{attribute 'linkalways'} 
{attribute 'no_explicit_call' := 'This FB is a CLASS and must be accessed using methods or properties'}
{attribute 'enable_dynamic_creation'}
FUNCTION_BLOCK OutputPort EXTENDS Disposable IMPLEMENTS I_OutputPort
VAR
	_name : T_MAXSTRING;
	_data : I_Datatype;
	parent : I_HaveOutputPorts;
	eventEmitter : EventEmitter;
END_VAR

METHOD PUBLIC Accept
VAR_INPUT
	Visitor : I_OutputPortVisitor;
END_VAR
Visitor.VisitOutputPort(this^);
END_METHOD

PROPERTY PUBLIC Data : I_Datatype
GET
Data := _data;
END_GET
END_PROPERTY

METHOD Protected EmitOnOutputPortChangeEvent
VAR_INPUT
	PortChanged : I_OutputPort;
END_VAR
VAR
	pOutputPortChangeEvent : POINTER TO OutputPortChangedEvent;
END_VAR
pOutputPortChangeEvent := __NEW(OutputPortChangedEvent(TargetOutputPort := PortChanged));
eventEmitter.Emit('OnOutputPortChanged',pOutputPortChangeEvent^);
pOutputPortChangeEvent^.Dispose();
END_METHOD

METHOD FB_init : BOOL
VAR_INPUT
	bInitRetains : BOOL; // if TRUE, the retain variables are initialized (warm start / cold start)
	bInCopyCode : BOOL;  // if TRUE, the instance afterwards gets moved into the copy code (online change)
	Name : T_MAXSTRING;
	Data : I_Datatype;
	Parent : I_HaveOutputPorts;
END_VAR
_name := Name;
_data := Data;
RegisterWithParent(Parent);
END_METHOD

PROPERTY PUBLIC Name : T_MAXSTRING
GET
Name := _name;
END_GET
END_PROPERTY

METHOD PUBLIC OffEvent
VAR_INPUT
	EventName : T_MaxString;
	EventHandler : I_EventHandler;
END_VAR
eventEmitter.OffEvent(EventName, EventHandler);
END_METHOD

METHOD PUBLIC OnceEvent
VAR_INPUT
	EventName : T_MaxString;
	EventHandler : I_EventHandler;
END_VAR
eventEmitter.OnceEvent(EventName, EventHandler);
END_METHOD

METHOD PUBLIC OnEvent
VAR_INPUT
	EventName : T_MaxString;
	EventHandler : I_EventHandler;
END_VAR
eventEmitter.OnEvent(EventName, EventHandler);
END_METHOD

METHOD PUBLIC RegisterWithParent
VAR_INPUT
	Parent : I_HaveOutputPorts;
END_VAR
IF Parent = 0 THEN
	RETURN;
END_IF

THIS^.parent := Parent;
Parent.AddOutputPort(THIS^);
END_METHOD

METHOD PUBLIC SerializeWith
VAR_INPUT
	Serializer : I_Serializer;
END_VAR
Serializer.StartObject();
Serializer.AddKeyString('name',_name);
Serializer.Addkey('datatype');
_data.SerializeTypeWith(Serializer);
Serializer.AddkeyObject('value',_data);
Serializer.EndObject();
END_METHOD

END_FUNCTION_BLOCK

(* stored: Version 1.1.0.1, ProductVersion 3.1.4024.12
   POU OutputPort: Id {4c7e0bce-9eb0-0f6a-044f-6a3cfc8b783d}, SpecialFunc None
   Folder Constructor: Id {677256cd-e8af-081b-2804-5689f5f4149b}
   Folder Protected: Id {6f5f4b13-ef19-01e5-075e-0ea3b801d3d7}
   Method Accept: Id {685a8b40-a5b2-0491-3a06-acbf37dad5a1}
   Property Data: Id {f88ed905-c54b-4c6d-be97-9339266743b0}
   Get Get: Id {120b55e4-6686-441d-ae9a-fc15e5629d7f}
   Method EmitOnOutputPortChangeEvent: Id {4cedd9f2-3d84-035e-18ce-b7ebc3af2524}
   Method FB_init: Id {1ba1d2d7-341d-0e8e-05ef-f5346255db4e}
   Property Name: Id {a6251d93-37b5-06d7-00eb-bc1261f23075}
   Get Get: Id {66530c4b-9811-0535-0d83-3db73e2195f3}
   Method OffEvent: Id {5f0c98a6-efae-06ce-0d53-00d24017a360}
   Method OnceEvent: Id {33aa55e6-cc64-0804-1f68-fe127e9ffd59}
   Method OnEvent: Id {83584882-e2df-000f-0211-5ef5ee02b990}
   Method RegisterWithParent: Id {c7baf534-bf05-4f66-b2b4-ef8e09f96124}
   Method SerializeWith: Id {dde3cc20-8117-4526-a740-816620bcd3a1} *)
